//-----------------------------------------------------------------------------------------------------
//																
//									 	Tkmatik sp z o.o.
//
//	Name					:		FB_Save
//	Author					:		AM
//	Release Date			:		12.01.2022
//	Current ver				:		v 0.1
// 	Last correction 		:		12.01.2022
// 
//	Description				:
//		Special FB for saving structures to CSV files						
//
//	Requared hardware		:
//
// 	Configuration			:
//
//
//-----------------------------------------------------------------------------------------------------

FUNCTION_BLOCK FB_RecipeSaveCSV

VAR_INPUT
	bExecute							: BOOL := FALSE;(* Rising edge starts program execution *)
	sFilePath							: T_MaxString;(* CSV destination file path and name *)
//	database							: POINTER TO STRING(255);	
	nRows          						: UDINT;                // Liczba wierszy
    nCols          						: UDINT; 
	database							: POINTER TO STRING(255);//ARRAY[0..MAX_PARAMS_VARIABLES_COUNT-1] OF STRING(255);
END_VAR
VAR CONSTANT
	MAX_CSV_FIELD_LENGTH				: UDINT	:= 255;	
END_VAR
VAR_IN_OUT
END_VAR

VAR
	
	sNetId			: T_AmsNetId := '';	(* TwinCAT system network address *)
	sCSVLine		: T_MaxString := '';(* Single CSV text line (row, record), we are using string as record buffer (your are able to see created fields) *)
	sCSVField		: T_MaxString := '';(* Single CSV field value (column, record field) *)
	nRow	 		: UDINT 	:= 0;(* Row number (record) *)
	nColumn			: UDINT 	:= 0;(* Column number (record field) *)
	hFile			: UINT		:= 0;(* File handle of the source file *)
	step			: DWORD 	:= 0;
	fbFileOpen		: FB_FileOpen;(* Opens file *)
	fbFileClose		: FB_FileClose;(* Closes file *)
	fbFilePuts		: FB_FilePuts;(* Writes one record (line) *)
	fbWriter		: FB_CSVMemBufferWriter;(* Helper function block used to create CSV data bytes (single record line) *)
	rtExecute		:	R_TRIG;                         //	Rtrig for start



END_VAR
VAR_OUTPUT                                                                                  
	bBusy												:	BOOL;                           //	FB is Busy
	bDone												:	BOOL;                           //	Load cycle done, DATA actual 
	bError												:	BOOL;                           //	Flag error
	nErrId												:	UDINT;                          //	Error ID
END_VAR

rtExecute(CLK:=bExecute);
IF (NOT bExecute) THEN
	bDone												:=	FALSE;
END_IF

CASE step OF
	0:	(* Wait for rising edge at bWrite variable *)
		IF rtExecute.Q THEN
			bBusy 	:= TRUE;
			bError	:= FALSE;
			nErrId	:= 0;
			hFile	:= 0;
			nRow	:= 0;
			nColumn	:= 0;
			step 	:= 1;
		END_IF

	1:	(* Open source file *)
		fbFileOpen(  bExecute := FALSE  );
		fbFileOpen( sNetId := sNetId, sPathName := sFilePath, nMode := FOPEN_MODEWRITE OR FOPEN_MODETEXT,(* Open file in TEXT mode! *)
					ePath := PATH_GENERIC, bExecute := TRUE );
		step := 2;

	2:(* Wait until open not busy *)
		fbFileOpen( bExecute := FALSE, bError => bError, nErrID => nErrID, hFile => hFile );
		IF NOT fbFileOpen.bBusy THEN
			IF NOT fbFileOpen.bError THEN
				step := 3;
			ELSE(* Error: file not found? *)
				step := 100;
			END_IF
		END_IF

	3:(* Convert one PLC record to CSV format *)
		sCSVLine := '';
		fbWriter.eCmd := eEnumCmd_First;(* Write first field value *)
		IF nRow <= nRows THEN

			FOR nColumn := 0 TO nCols BY 1 DO
 
				sCSVField := STRING_TO_CSVFIELD( database[ nRow ], FALSE );(* TODO: Get field value from your application *)

				(* Add new field to the record buffer *)
				fbWriter( 	pBuffer := ADR( sCSVLine ), cbBuffer := SIZEOF( sCSVLine ) - 1, putValue := sCSVField, pValue := 0, cbValue := 0,
							bCRLF := ( nColumn = nCols ) );(* bCRLF == TRUE => Write CRLF after the last field value *)
				IF fbWriter.bOk THEN
					fbWriter.eCmd := eEnumCmd_Next;(* Write next field value *)
				ELSE(* Error *)
					step := 100;
					RETURN;
				END_IF

			END_FOR(* FOR nColumn := 0... *)

			(* FB_FilePuts adds allready CR (carriage return) to the written line.
			We have to replace the $R$L characters with $L character to avoid double CR. *)
			IF RIGHT( sCSVLine, 2 ) = '$R$L' THEN
				sCSVLine := REPLACE( sCSVLine, '$L', 2, LEN( sCSVLine ) - 1 );
			END_IF

			nRow := nRow + 1;(* Increment number of created records (rows) *)
			step := 4;(* Write record to the file *)

		ELSE(* All rows written => Close file *)
			step := 10;
		END_IF

	4:	(* Write single text line *)
		fbFilePuts( bExecute := FALSE );
		fbFilePuts( sNetId := sNetId, hFile := hFile, sLine := sCSVLine, bExecute := TRUE );
		step := 5;

	5:(* Wait until write not busy *)
		fbFilePuts( bExecute := FALSE, bError => bError, nErrID => nErrID );
		IF NOT fbFilePuts.bBusy THEN
			IF NOT fbFilePuts.bError THEN
				step := 3;(* Write next record *)
			ELSE(* Error *)
				step := 100;
			END_IF
		END_IF

	10:	(* Close source file *)
		fbFileClose( bExecute := FALSE );
		fbFileClose( sNetId := sNetId, hFile := hFile, bExecute := TRUE );
		step := 11;

	11:(* Wait until close not busy *)
		fbFileClose( bExecute := FALSE, bError => bError, nErrID => nErrID );
		IF ( NOT fbFileClose.bBusy ) THEN
			bDone	:= TRUE;
			hFile := 0;
			step := 100;
		END_IF

	100: (* Error or ready step => cleanup *)
		IF ( hFile <> 0 ) THEN
			step := 10; (* Close the source file *)
		ELSE
			bBusy := FALSE;
			step := 0;	(* Ready *)
		END_IF

END_CASE

END_FUNCTION_BLOCK

(* stored: Version 1.1.0.1, ProductVersion 3.1.4026.13, FileIdentifier 59d98df1757a5f2f77cd22ec66ba06d097983a0e, FileSignature 212cd31aa44ffe37020c3cdb26922d2ca3d450250f71bea9dae2de1f2becaf31ea540e4e2a6e1afcb5b500d301392c9f792a72b3ad4cf53e4b3e6a94f213043a41c14c9691da9ec51548b083268926420e2b66b7abab002fc1f081d9c898145986651f529338c30e169a07f0689a09e73150603c140a7ab363fc389ace8ba6eeed0723acccfd106a46d48f6b7917f4a37b31aae726a8d57770321dd716f617481f38b60c36b89b665d6c21ad4597c9a8a703a7b99d0a97d106d9c0f13c4694266f01bfc50d91bd7b2eec32c249ee3735edb8544d47950eea052be6c2dde278c3e80b0faa24a51687bb4d62376f596edaa6ebd58cc21eb4d7ef5a433beaa2c16d
   POU FB_RecipeSaveCSV: Id {d65203d5-09ea-4c19-863d-a01b972c0703}, SpecialFunc None *)
